// TIA Portal V18 export
DATA_BLOCK "03_FDBACK_RAW"   // DB5, F_DB
{ S7_Optimized_Access := 'TRUE'; DB_Accessible_From_OPC_UA := 'FALSE' }
VERSION : 0.1
// stored: AutoNumber true, DBAccessibleFromOPCUA false, DBAccessibleFromWebserver true
   VAR
      AlwaysFALSE : Bool;
      AlwaysTRUE : Bool;
      "No Operation" : Bool;
      "Contactor Feedback Error [ =S1+PC1.CC1-Q66401..2 ]" : Bool;
      "Contactor Feedback Error [ =S1+PC1.CC1-X80201 ]" : Bool;
      "Contactor Feedback Error [ =S1+PC1.CC1-Q80001 ]" : Bool;
      "Contactor Feedback Error [ =S2+PC2.CC1-Q66401..2 ]" : Bool;
      "Contactor Feedback Error [ =S2+PC2.CC1-X80201 ]" : Bool;
      "Contactor Feedback Error [ =S2+PC2.CC1-Q80001 ]" : Bool;
   END_VAR
BEGIN
END_DATA_BLOCK
